TYPE ST_HMIData :
STRUCT
	s_Type			: STRING(12);
	s_Name			: STRING(25);
	r_Data			: REAL;
	s_Unit			: STRING(3);
END_STRUCT
END_TYPE

(* stored: Version 1.1.0.1, ProductVersion 3.1.4024.12
   DUT ST_HMIData: Id {ab4ca2da-3400-458a-9d4c-f812c0b50b5c} *)
